TYPE DUT_STRUCT_C000012_DEV :
STRUCT
	sCellName			:STRING := 'C000012';
	sIpAddress			:STRING := '';
	sAmsNetId			:STRING := '';
	sOpcUaURL			:STRING := 'opc.tcp://:4840';
	sStation1			:STRING := 'S000010';
END_STRUCT
END_TYPE

(* stored: Version 1.1.0.1, ProductVersion 3.1.4024.5
   DUT DUT_STRUCT_C000012_DEV: Id {127a6d39-2916-40f0-a9d7-dc35ea2e4c6d} *)
